TYPE ST_PROCESS_LIST_RESULT :
STRUCT
  wState    : WORD;   // wState == 0 --> all ok
  nIndex    : ULINT;
  stData    : ST_PROCESS_DATA;  // copy of list entry
END_STRUCT
END_TYPE

(* stored: Version 1.1.0.1
   DUT ST_PROCESS_LIST_RESULT: Id {7a3f0ad8-7076-46b9-b446-1a9360c14ec2} *)
